FUNCTION_BLOCK eIX (* Input service interface function block for boolean input data with event-base trigger *)
  (* Standard: 61499-2; Description: Copyright (c) 2025 Maximilian Scharf This program and the accompanying materials are made available under the terms of the Eclipse Public License 2.0 which is available at https://www.eclipse.org/legal/epl-2.0/ SPDX-License-Identifier: EPL-2.0 *)
  (* Version 3.0, 2025-04-14, Franz Höpfinger, HR Agrartechnik GmbH, Made Version 3.0.0 inspired by Work from Patrick Aigner *)
  (* Version 1.0, 2025-05-05, Maximilian Scharf *)
  PACKAGE eclipse4diac::io::eio;
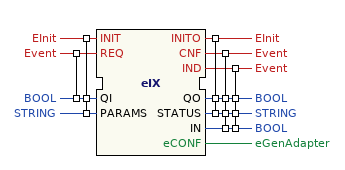
  EVENT_INPUT
    INIT : EInit WITH QI, PARAMS; (* Service Initialization *)
    REQ WITH QI; (* Service Request *)
  END_EVENT
  EVENT_OUTPUT
    INITO : EInit WITH QO, STATUS; (* Initialization Confirm *)
    CNF WITH QO, STATUS, IN; (* Confirmation of Requested Service *)
    IND WITH QO, STATUS, IN; (* Indication from Resource *)
  END_EVENT
  VAR_INPUT
    QI : BOOL; (* Event Input Qualifier *)
    PARAMS : STRING; (* Service Parameters *)
  END_VAR
  VAR_OUTPUT
    QO : BOOL; (* Event Output Qualifier *)
    STATUS : STRING; (* Service Status *)
    IN : BOOL; (* Input data from resource *)
  END_VAR
  PLUGS
    eCONF : eclipse4diac::io::eio::eGenAdapter; (* Configuration of Event-based-Trigger *)
  END_PLUGS
END_FUNCTION_BLOCK
